Fanuc KAREL source: kx00013.KL

-- PROVISIONAL review KL for V940-1; original PC SHA256 d45c01971e638aba87cb1948e7aa2f28ee6c57e4b0823a9fbc145e8834c8ce31
-- Incomplete behavior may be omitted. Consult companion uncertainty JSON. Do not deploy.
PROGRAM KX00013
%NOLOCKGROUP
VAR
  I : INTEGER
  J : INTEGER
  B : BOOLEAN
  F : FILE
  S : STRING[80]
-- UNRESOLVED_DECL P type=000102
BEGIN
  -- V9_ZERO_TABLE_METADATA_HINT layout=0001; no indexed target words; source/name/runtime held
  -- UNRESOLVED_PC offsets 5-7; opcodes 9C,4E
  -- UNRESOLVED_PC offsets 12-16; opcodes 7F
END KX00013
